FUNCTION_BLOCK automaticoPreparadorPolimero (* Basic Function Block Type *)
  (* Standard: 61499-2 *)
  (* Version 0.0, 09/04/2026, Template *)
  PACKAGE Hidryco.HidrycoLib;
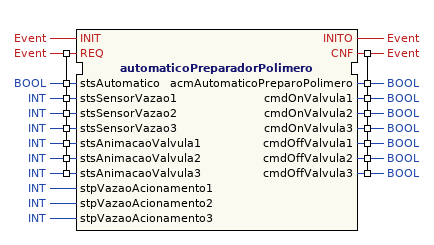
  EVENT_INPUT
    INIT; (* Initialization Request *)
    REQ WITH stsSensorVazao1, stsSensorVazao2, stsSensorVazao3, stsAnimacaoValvula1, stsAnimacaoValvula2, stsAnimacaoValvula3, stsAutomatico; (* Normal Execution Request *)
  END_EVENT
  EVENT_OUTPUT
    INITO; (* Initialization Confirm *)
    CNF WITH acmAutomaticoPreparoPolimero, cmdOnValvula1, cmdOnValvula2, cmdOnValvula3, cmdOffValvula1, cmdOffValvula2, cmdOffValvula3; (* Execution Confirmation *)
  END_EVENT
  VAR_INPUT
    stsAutomatico : BOOL;
    stsSensorVazao1 : INT;
    stsSensorVazao2 : INT;
    stsSensorVazao3 : INT;
    stsAnimacaoValvula1 : INT;
    stsAnimacaoValvula2 : INT;
    stsAnimacaoValvula3 : INT;
    stpVazaoAcionamento1 : INT;
    stpVazaoAcionamento2 : INT;
    stpVazaoAcionamento3 : INT;
  END_VAR
  VAR_OUTPUT
    acmAutomaticoPreparoPolimero : BOOL;
    cmdOnValvula1 : BOOL;
    cmdOnValvula2 : BOOL;
    cmdOnValvula3 : BOOL;
    cmdOffValvula1 : BOOL;
    cmdOffValvula2 : BOOL;
    cmdOffValvula3 : BOOL;
  END_VAR
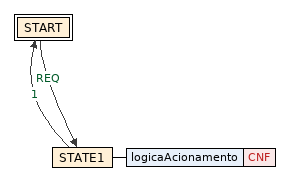
  EC_STATES
    START; (* Initial State *)
    STATE1 : logicaAcionamento -> CNF;
  END_STATES
  EC_TRANSITIONS
    START TO STATE1 := REQ;
    STATE1 TO START := 1;
  END_TRANSITIONS
  ALGORITHM INIT IN ST: (* Initialization algorithm *)
;
  END_ALGORITHM
  ALGORITHM REQ IN ST: (* Normally executed algorithm *)
;
  END_ALGORITHM
  ALGORITHM logicaAcionamento IN ST:
IF stsAutomatico THEN
    IF stsSensorVazao1 > stpVazaoAcionamento1 THEN
        cmdOnValvula1  := TRUE;
        cmdOffValvula1 := FALSE;
    ELSE
        cmdOnValvula1  := FALSE;
        cmdOffValvula1 := TRUE;
    END_IF;

    (* Válvula 2 *)
    IF stsSensorVazao2 > stpVazaoAcionamento2 THEN
        cmdOnValvula2  := TRUE;
        cmdOffValvula2 := FALSE;
    ELSE
        cmdOnValvula2  := FALSE;
        cmdOffValvula2 := TRUE;
    END_IF;

    (* Válvula 3 *)
    IF stsSensorVazao3 > stpVazaoAcionamento3 THEN
        cmdOnValvula3  := TRUE;
        cmdOffValvula3 := FALSE;
    ELSE
        cmdOnValvula3  := FALSE;
        cmdOffValvula3 := TRUE;
    END_IF;
ELSE
    cmdOnValvula1  := FALSE;
    cmdOnValvula2  := FALSE;
    cmdOnValvula3  := FALSE;
    cmdOffValvula1 := FALSE;
    cmdOffValvula2 := FALSE;
    cmdOffValvula3 := FALSE;
END_IF;

acmAutomaticoPreparoPolimero :=
    stsAutomatico AND
    (
        (stsAnimacaoValvula1 = 1) OR
        (stsAnimacaoValvula2 = 1) OR
        (stsAnimacaoValvula3 = 1)
    );
;
  END_ALGORITHM
END_FUNCTION_BLOCK
